FUNCTION_BLOCK OPCUA_BOOL_VARIABLE_LISTENER
  {SET_ATTRIBUTE(OpcUa, DEVICE.SENSOR)}
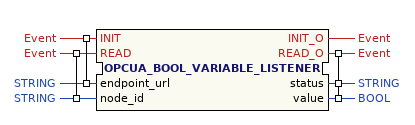
  EVENT_INPUT
    INIT WITH endpoint_url;
    READ WITH node_id; {SET_ATTRIBUTE(OpcUa, Method)}
  END_EVENT
  EVENT_OUTPUT
    INIT_O;
    READ_O WITH status, value;
  END_EVENT
  VAR_INPUT
    endpoint_url : STRING; {SET_ATTRIBUTE(OpcUa, Constant)}
    node_id : STRING; {SET_ATTRIBUTE(OpcUa, Variable)}
  END_VAR
  VAR_OUTPUT
    status : STRING; {SET_ATTRIBUTE(OpcUa, Variable)}
    value : BOOL; {SET_ATTRIBUTE(OpcUa, Variable)}
  END_VAR
END_FUNCTION_BLOCK
